(* Logix 5000 project; controller test vendor 1 type 14 code 196 rev 35.11; software revision 35.00 *)

TASK MainTask (continuous, watchdog 500 ms) : MainProgram

MODULES
   Local : vendor 1 type 14 code 196 (5069 0, rev 35.11)
END_MODULES

PROGRAM MainProgram   (* main routine MainRoutine *)
VAR
   Arm_Pressure_Switch : BOOL;
   Arm_Speed_Percentage : REAL;
   Box_in_position : BOOL;
   Box_On_Conveyor_belt : BOOL;
   Emergency_Stop : BOOL;
   Enable_Conveyor_Belt : BOOL;
   Enable_Robotic_Arm : BOOL;
   Label_Reader : BOOL;
   Limit_Switch : BOOL;
   Percentage_Arm_Force : REAL;
   Running : BOOL;
   Start_Button : BOOL;
END_VAR

ROUTINE MainRoutine   (* ladder *)
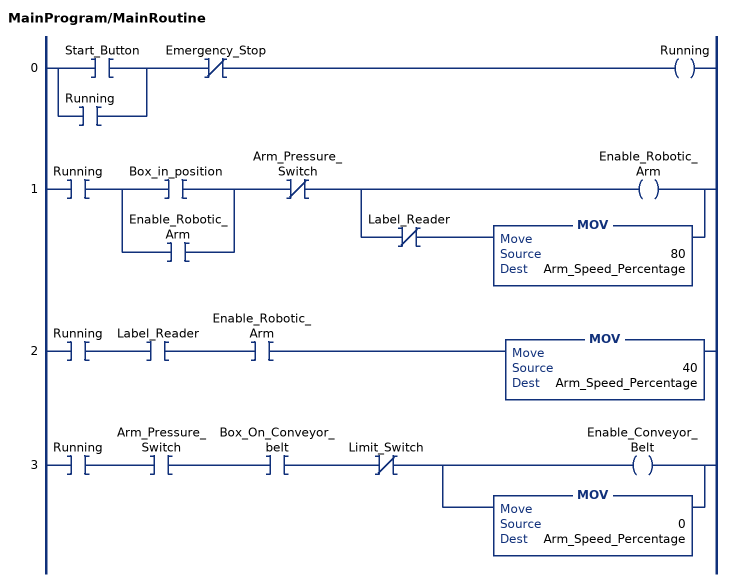
   0: [XIC(Start_Button) ,XIC(Running) ]XIO(Emergency_Stop)OTE(Running);
   1: XIC(Running)[XIC(Box_in_position) ,XIC(Enable_Robotic_Arm) ]XIO(Arm_Pressure_Switch)[OTE(Enable_Robotic_Arm) ,XIO(Label_Reader) MOV(80,Arm_Speed_Percentage) ];
   2: XIC(Running)XIC(Label_Reader)XIC(Enable_Robotic_Arm)MOV(40,Arm_Speed_Percentage);
   3: XIC(Running)XIC(Arm_Pressure_Switch)XIC(Box_On_Conveyor_belt)XIO(Limit_Switch)[OTE(Enable_Conveyor_Belt) ,MOV(0,Arm_Speed_Percentage) ];
END_ROUTINE
END_PROGRAM
